TYPE ST_ElementMasterSlave :
(**************************************************************************************
 * 	Application		:	BoxControl Framework
 *	Revision		:	$Revision: 404529 $
 *	Revision date	:	$Date: 2018-04-23 08:21:38 +0200 (Mo., 23 Apr 2018) $
 *	Last changed by	:	$Author: b7bolm $
 *	URL				:	$URL: http://almscdc.swisslog.com/repo/SWPD/Development/BoxControlFramework/20_Release/trunk/01_Software/BCF/BCF/JumpStart/20_Product/10_App/13_Elements/10_Lib/10_Conv/01_DUTs/ST_ElementMasterSlave.TcDUT $
 *
 *	Purpose			:	Master slave info
 *
 * ------------------------------------------------------------------------------------
 *	Copyright Swisslog [IP AG], Switzerland. All rights reserved.
 * 
 * ------------------------------------------------------------------------------------
 *	
 * 	Revision History: 
 *
 * 	VERSION			DATE			INITIALS			DESCRIPTION
 *	0.1				01.01.2001		swl					Example
 *
 **************************************************************************************)
STRUCT
	Master		: ST_ElementMasterSlaveEntry;
	Slave		: ST_ElementMasterSlaveEntry;
	Master_12	: ST_ElementMasterSlaveEntry;
	Slave_12	: ST_ElementMasterSlaveEntry;
	Master_34	: ST_ElementMasterSlaveEntry;
	Slave_34	: ST_ElementMasterSlaveEntry;

END_STRUCT
END_TYPE

(* stored: Version 1.1.0.1, ProductVersion 3.1.4022.12
   DUT ST_ElementMasterSlave: Id {517691c7-3c70-4901-9903-962e3e3c6ad8} *)
